{attribute 'qualified_only'}
TYPE E_PML_Command :
(
	Undefined := 0,	// 0
	Reset,			// 1
	Start,			// 2
	Stop,			// 3
	Hold,			// 4
	Unhold,			// 5
	Suspend,		// 6
	Unsuspend,		// 7
	Abort,			// 8
	Clear,			// 9
	Complete		// 10
) UINT;
END_TYPE

(* stored: Version 1.1.0.1, ProductVersion 3.1.4024.5
   DUT E_PML_Command: Id {d58dcc90-7cdb-4070-848b-5ff73f550e6f} *)
